// TwinCAT 3 PLC project _01_Simple
// ProgramVersion: 3.1.4026.18
// libraries:
//   Tc2_Standard, * (Beckhoff Automation GmbH)
//   Tc2_System, * (Beckhoff Automation GmbH)
//   Tc2_Utilities, * (Beckhoff Automation GmbH)
//   StageCore, * (_)
//   StageUtils, * (_)
// project tree:
//   01_Entities/01_ToggleExample/ I_Toggle.TcIO, Toggle.TcPOU, ToggleExample.TcPOU
//   01_Entities/ EntitiesExample.TcPOU
//   02_Jobs/ JobsExample.TcPOU
//   02_Jobs/01_CountTo/ CountToJob.TcPOU (not stored), CountToExample.TcPOU, MyWorker.TcPOU (not stored)
//   04_Broadcast/ BroadcastExample.TcPOU
//   04_Broadcast/Safety/ Safety.TcPOU, SafetyExample.TcPOU, StoppableEntity.TcPOU
//   / PlcTask.TcTTO
//   00_MAIN/ MAIN.TcPOU
//   03_States/01_PackML/ ExampleStateMachine.TcPOU (not stored), PackMLExample.TcPOU, StateContext.TcDUT (not stored)
//   03_States/01_PackML/States/ StateAborted.TcPOU (not stored), StateComplete.TcPOU (not stored), StateExecute.TcPOU (not stored), StateHeld.TcPOU, StateIdle.TcPOU, StateStopped.TcPOU (not stored), StateSuspended.TcPOU, _AbstractState.TcPOU (not stored)
//   03_States/ StatesExample.TcPOU
// real-time tasks:
//   TASK PlcTask: cycle T#10ms, priority 20, ADS port 350
//   TASK PlcTask1: cycle T#10ms, priority 21, ADS port 351

CONFIGURATION _01_Simple
    RESOURCE PLC ON TwinCAT3
        TASK PlcTask(INTERVAL := T#10ms, PRIORITY := 20);
        PROGRAM MAIN WITH PlcTask : MAIN;
    END_RESOURCE
END_CONFIGURATION

// ---- 01_Entities/01_ToggleExample/I_Toggle.TcIO
INTERFACE I_Toggle EXTENDS I_RawComponent

PROPERTY IsOn : BOOL
GET
END_GET
END_PROPERTY

METHOD SwitchOff
VAR_INPUT
END_VAR
END_METHOD

METHOD SwitchOn
VAR_INPUT
END_VAR
END_METHOD

PROPERTY Tag : I_Tag
GET
END_GET
END_PROPERTY

METHOD Toggle
VAR_INPUT
END_VAR
END_METHOD

END_INTERFACE

// ---- 00_MAIN/MAIN.TcPOU
PROGRAM MAIN
VAR
END_VAR

Runtime();

EntitiesExample();
JobsExample();
StatesExample();
BroadcastExample();

END_PROGRAM

// ---- 01_Entities/EntitiesExample.TcPOU
PROGRAM EntitiesExample
VAR
END_VAR

ToggleExample();

END_PROGRAM

// ---- 01_Entities/01_ToggleExample/ToggleExample.TcPOU
PROGRAM ToggleExample
VAR
	livingroom: Toggle;
	stairway: ARRAY[1..2] OF Toggle;
	kitchen: Toggle;
	bedroom: Toggle;
	
	cmd: (_SwitchOn, _SwitchOff, _Toggle) := _Toggle; // What you want to do?
	sRoomToCmd: Str := '*.bedroom'; // Who is the target?
	bRun: BOOL; // Rising edge will trigger the state change.
	
	iEtt: I_Entity;
	iComp: I_Component;
	iToggle: I_Toggle;
	
END_VAR

IF bRun THEN
	bRun := FALSE;
	
	WHILE IsOk(GetNextEntity(iEtt)) DO
		iComp := 0;
		
		WHILE IsOk(iEtt.GetNextComp(iComp)) DO
			IF NOT __QUERYINTERFACE(iComp.Raw, iToggle) THEN
				CONTINUE;
			END_IF
			
			IF IsOk(MatchPath(iToggle.Tag.Id, sRoomToCmd)) THEN
				CASE cmd OF
					_SwitchOn:
						iToggle.SwitchOn();
						
					_SwitchOff:
						iToggle.SwitchOff();
						
					_Toggle:
						iToggle.Toggle();
						
				END_CASE
			END_IF
			
			EXIT;
		END_WHILE
	END_WHILE
END_IF

END_PROGRAM

// ---- 01_Entities/01_ToggleExample/Toggle.TcPOU
FUNCTION_BLOCK Toggle IMPLEMENTS I_Toggle
VAR_INPUT
END_VAR
VAR_OUTPUT
END_VAR
VAR
	_ett: EntityStart;
		_component: Component(THIS^);
		_tag: Tag;
	_ettEnd: EntityEnd;
	
	_bValue: BOOL;
END_VAR

PROPERTY IsOn : BOOL
GET
IsOn := _bValue;
END_GET
END_PROPERTY

METHOD SwitchOff
_bValue := FALSE;
END_METHOD

METHOD SwitchOn
_bValue := TRUE;
END_METHOD

PROPERTY Tag : I_Tag
GET
Tag := _tag;
END_GET
END_PROPERTY

METHOD Toggle
_bValue := NOT _bValue;
END_METHOD

END_FUNCTION_BLOCK

// ---- 02_Jobs/JobsExample.TcPOU
PROGRAM JobsExample
VAR
END_VAR

CountToExample();

END_PROGRAM

// ---- 02_Jobs/01_CountTo/CountToExample.TcPOU
PROGRAM CountToExample
VAR
	// An array of jobs to do
	myWorker: MyWorker;
	counting: ARRAY[1..10] OF CountToJob := [(CountTo := 200, Worker := myWorker.Base)];
	i: UDINT;
	
	// Rising edge will trigger the state change.
	bStart: BOOL;
END_VAR

IF bStart THEN
	bStart := FALSE;
	FOR i := 1 TO 10 DO
	counting[i].Start();
	END_FOR	
	
END_IF

END_PROGRAM

// ---- 03_States/StatesExample.TcPOU
PROGRAM StatesExample
VAR
END_VAR

PackMLExample();

END_PROGRAM

// ---- 03_States/01_PackML/PackMLExample.TcPOU
PROGRAM PackMLExample
VAR
	example: ExampleStateMachine;
	
	iStateResult: I_State;
	iSmgr: I_StateManager;
	bError: BOOL;
	bInit: BOOL := TRUE;
	
	
	sStateToRequest: Str := '*.idle'; // Use this variable to tell program which state to request
	bRequest: BOOL; // Rising edge will trigger the state change.
	
END_VAR

IF bInit THEN
	bInit := FALSE;
	bError := IsFail(GetStateManager(example.Entity, iSmgr));
END_IF

IF bError THEN
	RETURN;
END_IF

IF NOT bRequest THEN
	RETURN;
END_IF

bRequest := FALSE;

IF IsOk(GetState(example.Entity, sStateToRequest, iStateResult)) THEN
	iSmgr.Request(iStateResult);
END_IF

END_PROGRAM

// ---- 04_Broadcast/BroadcastExample.TcPOU
PROGRAM BroadcastExample
VAR
END_VAR

SafetyExample();

END_PROGRAM

// ---- 04_Broadcast/Safety/SafetyExample.TcPOU
PROGRAM SafetyExample
VAR
	stoppable: ARRAY[1..20] OF StoppableEntity;
	safety: Safety;
END_VAR

END_PROGRAM

// ---- 04_Broadcast/Safety/StoppableEntity.TcPOU
FUNCTION_BLOCK StoppableEntity IMPLEMENTS I_Callable
VAR_INPUT
END_VAR
VAR_OUTPUT
END_VAR
VAR
	_ett: EntityStart;
		_onSafetyStop: Receiver := (Callable := THIS^);
	_ettEnd: EntityEnd;

	_bSafetyStopLock: BOOL;
END_VAR

(*
This method provides a standardized way for other objects to interact with the object that owns it.
*)
METHOD Call
VAR_INPUT
	iArg	: StageCore.I_Arg;
END_VAR
VAR
	iSafetyStopState: I_BoolArg;
END_VAR
IF IsOk(IArgToIBoolArg(iArg, iSafetyStopState)) THEN
	_bSafetyStopLock := iSafetyStopState.Get;
END_IF
END_METHOD

END_FUNCTION_BLOCK

// ---- 04_Broadcast/Safety/Safety.TcPOU
FUNCTION_BLOCK Safety IMPLEMENTS I_Execute, I_Init
VAR
	_exe: Execute(THIS^);
	_init: Init(THIS^);	

	_bSafetyStopState: BOOL;
	_rtSafetyStop: R_TRIG;
	_ftSafetyStop: F_TRIG;
	
	_ett: EntityStart;
		_safetyStop: Signal;
	_ettEnd: EntityEnd;
END_VAR

(*
If registered, this method will be executed cyclically.
*)
METHOD Execute
VAR_INPUT
	nPhase	: INT;
END_VAR
VAR
	_safetyStopState: BoolArg(_bSafetyStopState);
END_VAR
_rtSafetyStop(CLk := _bSafetyStopState);
_ftSafetyStop(CLk := _bSafetyStopState);

IF _rtSafetyStop.Q OR _ftSafetyStop.Q THEN
	
	_safetyStop.Emit(_safetyStopState);
END_IF
END_METHOD

(*
If registered, this method will be executed upon startup.
*)
METHOD Init
VAR_INPUT
	nPhase	: INT;
END_VAR
VAR
	iEtt: I_Entity;
	iRec: I_Receiver;
END_VAR
WHILE IsOk(GetNextEntity(iEtt)) DO
	IF IsOk(GetReceiver(iEtt, '*._onSafetyStop.*', iRec)) THEN
		_safetyStop.Pair(iRec);
	END_IF
END_WHILE
END_METHOD

END_FUNCTION_BLOCK

// ---- 03_States/01_PackML/States/StateHeld.TcPOU
FUNCTION_BLOCK StateHeld EXTENDS _AbstractState
VAR_INPUT
END_VAR
VAR_OUTPUT
END_VAR
VAR
	_ton: TON;
END_VAR

(*
Determines whether the state can be activated.  
Returns `TRUE` by default but can be overridden for specific activation conditions.
*)
METHOD PROTECTED CanActivate : BOOL
CanActivate := _ctx.smgr.Current.Tag = _ctx.execute.Tag;
END_METHOD

(*
Executed when the state is entered.  
Provides a hook for defining state-specific behavior to be performed during the transition into this state.
*)
METHOD PROTECTED OnEntry
_ton(IN := FALSE);
END_METHOD

(*
Executed during the state's operation.  
Used to define state-specific logic that runs while the state is active.
*)
METHOD PROTECTED OnExecute
VAR
	strb: Strb;
END_VAR
_ton(IN := TRUE, PT := T#10S);
IF _ton.Q THEN
	_ctx.smgr.Request(_ctx.execute);
END_IF

_ctx.sHmiStatusText :=
	strb.Set('Held: Smoke break. Remaining time: ')
		.Append(Strf.SimpleTime(_ton.PT - _ton.ET, 'S', 'M'))
		.Read();
END_METHOD

END_FUNCTION_BLOCK

// ---- 03_States/01_PackML/States/StateIdle.TcPOU
FUNCTION_BLOCK StateIdle EXTENDS _AbstractState
VAR_INPUT
END_VAR
VAR_OUTPUT
END_VAR
VAR
END_VAR

(*
Determines whether the state can be activated.  
Returns `TRUE` by default but can be overridden for specific activation conditions.
*)
METHOD PROTECTED CanActivate : BOOL
VAR
	cmp: TagCmp;
END_VAR
CanActivate := cmp.Set(_ctx.smgr.Current.Tag)
					.Match(_ctx.stopped.Tag)
					.Match(_ctx.complete.Tag)
					.IsTrue();
END_METHOD

(*
Executed during the state's operation.  
Used to define state-specific logic that runs while the state is active.
*)
METHOD PROTECTED OnExecute
VAR
	strb: Strb;
END_VAR
_ctx.rLevel := _ctx.rLevel + 1;
IF _ctx.rLevel >= 600 THEN
	_ctx.smgr.Request(_ctx.execute);
END_IF

_ctx.sHmiStatusText :=
	strb.Set('Idle: Level - ')
		.Append(Strf.Fmt('%.0f', F_LREAL(_ctx.rLevel)))
		.Read();
END_METHOD

END_FUNCTION_BLOCK

// ---- 03_States/01_PackML/States/StateSuspended.TcPOU
FUNCTION_BLOCK StateSuspended EXTENDS _AbstractState
VAR_INPUT
END_VAR
VAR_OUTPUT
END_VAR
VAR
	_bSuspendLock: BOOL;
END_VAR

(*
Determines whether the state can be activated.  
Returns `TRUE` by default but can be overridden for specific activation conditions.
*)
METHOD PROTECTED CanActivate : BOOL
CanActivate := _ctx.smgr.Current.Tag = _ctx.execute.Tag;
END_METHOD

(*
Executed when the state is entered.  
Provides a hook for defining state-specific behavior to be performed during the transition into this state.
*)
METHOD PROTECTED OnEntry
_ctx.sHmiStatusText := 'Suspended: I guess we wait... ';
END_METHOD

END_FUNCTION_BLOCK
